// TIA Portal V21 export
TYPE "lubricationSystemOut"
   STRUCT
      pump1Start : Bool;
      pump2Start : Bool;
      heaterOn : Bool;
      waterVlvOpen : Bool;
      oilToCoolerVlv : Bool;
   END_STRUCT;
END_TYPE
